// TIA Portal project "Cooking Timer" (V17)
// Cooking Timer
// A microwave should run for 1 minute when the start button is turned ON.
// An additional 30 seconds should be added if a +30s button is turned ON.

(* hardware
DEVICE "S7-1200 station_1"  S7-1200 Station
   slot 0: "Rack_0"  S7-1200 Rack  Rack  V1.0
   slot 1: "PLC_1"  CPU 1212C AC/DC/Rly  6ES7 212-1BE40-0XB0  V4.5
*)

// ===== PLC "PLC_1"  CPU 1212C AC/DC/Rly =====

VAR_GLOBAL   // PLC tag table "Default tag table"
   "Start" AT %I0.0 : Bool;
   "+30S" AT %I0.1 : Bool;
   "Microwave" AT %I0.2 : Bool;
   "Tag_1" AT %M0.0 : Bool;
   "Tag_2" AT %M0.1 : Bool;
   "Tag_3" AT %M0.2 : Bool;
END_VAR

// folder: System blocks/Program resources

DATA_BLOCK "IEC_Timer_0_DB"   // DB1
{ S7_Optimized_Access := 'TRUE' }
AUTHOR : Simatic
FAMILY : IEC
NAME : IEC_TMR
VERSION : 1.0
// stored: InstanceOfName IEC_TIMER
"IEC_TIMER"
BEGIN
END_DATA_BLOCK

DATA_BLOCK "IEC_Timer_0_DB_1"   // DB2
{ S7_Optimized_Access := 'TRUE' }
AUTHOR : Simatic
FAMILY : IEC
NAME : IEC_TMR
VERSION : 1.0
// stored: InstanceOfName IEC_TIMER
"IEC_TIMER"
BEGIN
END_DATA_BLOCK

// folder: (top level)

ORGANIZATION_BLOCK "Main"   // OB1, LAD, ProgramCycle
TITLE = "Main Program Sweep (Cycle)"
{ S7_Optimized_Access := 'TRUE' }
VERSION : 0.1
   VAR_INPUT
      Initial_Call : Bool;   // Initial call of this OB
      Remanence : Bool;   // =True, if remanent data are available
   END_VAR
BEGIN

REGION Network 1
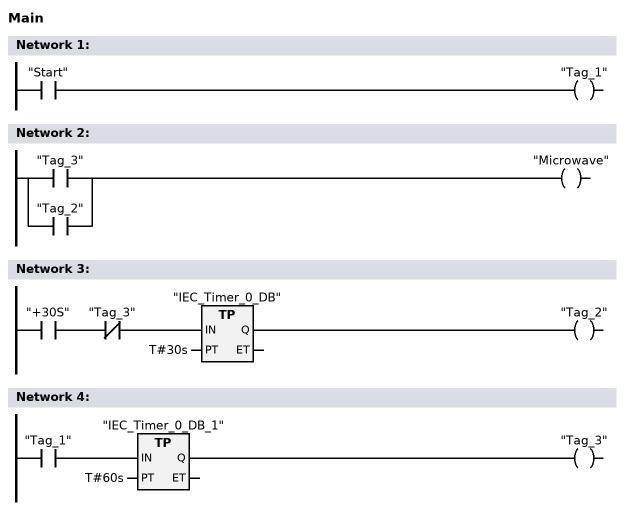
   RUNG wire#powerrail
      Contact( "Start" )
      Coil( "Tag_1" )
   END_RUNG
   // the same network as SCL:
   "Tag_1" := "Start";
END_REGION

REGION Network 2
   RUNG wire#powerrail
      Contact( "Tag_3" )
      wire#w1
      Coil( "Microwave" )
   END_RUNG
   RUNG wire#powerrail
      Contact( "Tag_2" )
   END_RUNG wire#w1
   // the same network as SCL:
   "Microwave" := "Tag_3" OR "Tag_2";
END_REGION

REGION Network 3
   "IEC_Timer_0_DB".TP(IN := "+30S" AND NOT "Tag_3", PT := T#30s);
   "Tag_2" := "IEC_Timer_0_DB".Q;
END_REGION

REGION Network 4
   "IEC_Timer_0_DB_1".TP(IN := "Tag_1", PT := T#60s);
   "Tag_3" := "IEC_Timer_0_DB_1".Q;
END_REGION
END_ORGANIZATION_BLOCK